// TIA Portal V16 export
// export: Created 2024-06-18T17:14:06.6356534Z, ExportSetting WithDefaults, DisplayName Totally Integrated Automation Portal, DisplayVersion V16, DisplayName TIA Portal Version Control Interface, DisplayVersion V16, DisplayName TIA Portal Openness, DisplayVersion V16, DisplayName STEP 7 Professional, DisplayVersion V16, DisplayName STEP 7 Safety, DisplayVersion V16, DisplayName WinCC Advanced, DisplayVersion V16
TYPE "Axis.RB_Memórias"
TITLE = Memorias do robô
// stored: IsFailsafeCompliant false
   STRUCT
      RB_Mem_Internas { S7_SetPoint := 'True'} : "Axis.RB_Memórias_Internas";   // Memórias Internas
      RB_Mem_Externas { S7_SetPoint := 'True'} : "Axis.RB_Memórias_Externas";   // Memórias Externas
   END_STRUCT;
END_TYPE
